# EPICS substitutions: hugo/source/db/Beckhoff_3XXX/ecmcEL3202-0010.substitutions
file "ecmc_analogInput-chX.template"
{
  pattern {CH_ID, ESLO, EOFF, EGU,    PREC}
          {01,    0.01, 0,    "DegC", 3   }
          {02,    0.01, 0,    "DegC", 3   }
}

file "ecmc_status-chX.template"
{
  pattern {CH_ID, KEY }
          {01,    "AI"}
          {02,    "AI"}
}
